// Mitsubishi GX Works2 project: 3Kolv   PLC: FX1S

// global labels: Global1
VAR_GLOBAL
  Start AT X006 : BOOL;
  Go AT M1 : BOOL;
  StopB AT X007 : BOOL;
  Cyl_1Inne AT X001 : BOOL;
  Cyl_1Ute AT X000 : BOOL;
  Cyl1_UT AT M2 : BOOL;
  Cyl_3Inne AT X005 : BOOL;
  Cyl_3Ute AT X004 : BOOL;
  Cyl3_UT AT M3 : BOOL;
  Cyl_3UT AT M5 : BOOL;
  Cyl1_IN AT M4 : BOOL;
  C3_STEG2 AT M6 : BOOL;
  Cyl3_IN AT M7 : BOOL;
  CTU_1 : CTU;
  Cyl1_Inåt AT Y000 : BOOL;
  Cyl1_Utåt AT Y001 : BOOL;
  Cyl3_Inåt AT Y004 : BOOL;
  Cyl3_Utåt AT Y005 : BOOL;
END_VAR

// task Task_01 (event TRUE, interval 0, priority 31): POU_01

PROGRAM POU_01
VAR
  Timer_Cyl3 : TON;
END_VAR
(* structured ladder/FBD written out as ST: instructions are called as NAME(EN, inputs, outputs); _pN, _eN, _tN stand for wires *)
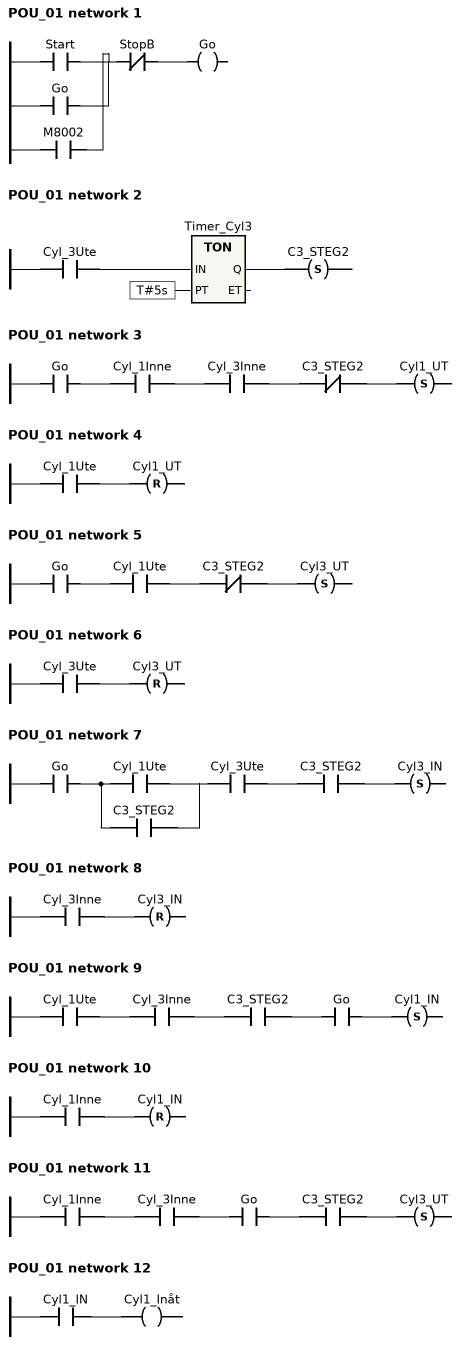
(* network 1 *)
Go := (Start OR Go OR M8002) AND NOT StopB;
(* network 2 *)
Timer_Cyl3(IN := Cyl_3Ute, PT := T#5s);
SET(Timer_Cyl3.Q, C3_STEG2);
(* network 3 *)
SET(Go AND Cyl_1Inne AND Cyl_3Inne AND NOT C3_STEG2, Cyl1_UT);
(* network 4 *)
RST(Cyl_1Ute, Cyl1_UT);
(* network 5 *)
SET(Go AND Cyl_1Ute AND NOT C3_STEG2, Cyl3_UT);
(* network 6 *)
RST(Cyl_3Ute, Cyl3_UT);
(* network 7 *)
SET((((Go AND Cyl_1Ute) OR (Go AND C3_STEG2)) AND Cyl_3Ute) AND C3_STEG2, Cyl3_IN);
(* network 8 *)
RST(Cyl_3Inne, Cyl3_IN);
(* network 9 *)
SET(Cyl_1Ute AND Cyl_3Inne AND C3_STEG2 AND Go, Cyl1_IN);
(* network 10 *)
RST(Cyl_1Inne, Cyl1_IN);
(* network 11 *)
SET(Cyl_1Inne AND Cyl_3Inne AND Go AND C3_STEG2, Cyl3_UT);
(* network 12 *)
Cyl1_Inåt := Cyl1_IN;
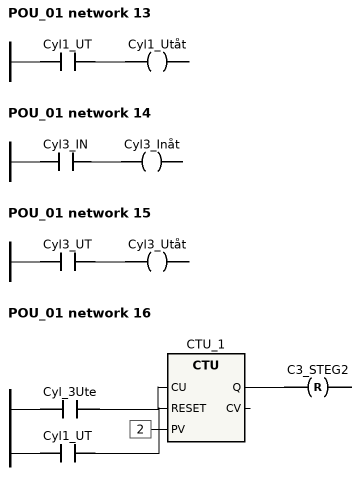
(* network 13 *)
Cyl1_Utåt := Cyl1_UT;
(* network 14 *)
Cyl3_Inåt := Cyl3_IN;
(* network 15 *)
Cyl3_Utåt := Cyl3_UT;
(* network 16 *)
CTU_1(CU := Cyl_3Ute, RESET := Cyl1_UT, PV := 2);
RST(CTU_1.Q, C3_STEG2);
END_PROGRAM
